% RSLogix 500 project PLCTEST_BAK000.RSS, saved by version 12.00.00.00 %
PROJECT "DRACO"    % processor: MicroLogix 1400 %

PROGRAM FILES
  LAD 2 "MAIN"  4 rungs
  LAD 3 "ALARM"  4 rungs
  LAD 4 "DIGITAL IO"  7 rungs
  LAD 5 "CONTROL"  6 rungs

DATA FILES
  O0 OUTPUT  7 elements
  I1 INPUT  10 elements
  S2 STATUS  66 elements
  B3 BINARY  1 elements
  T4 TIMER  3 elements
  C5 COUNTER  1 elements
  R6 CONTROL  1 elements
  N7 INTEGER  1 elements
  F8 FLOAT  1 elements

LADDER 2 "MAIN"
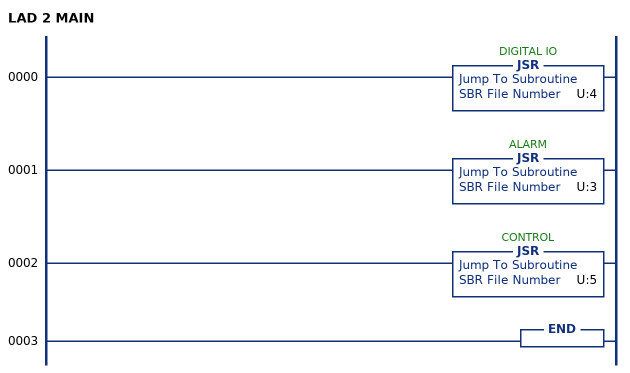
% Rung: 0 %
SOR JSR U:4 EOR
%   U:4  "DIGITAL IO" %
% Rung: 1 %
SOR JSR U:3 EOR
%   U:3  "ALARM" %
% Rung: 2 %
SOR JSR U:5 EOR
%   U:5  "CONTROL" %
% Rung: 3 %
SOR END EOR

LADDER 3 "ALARM"
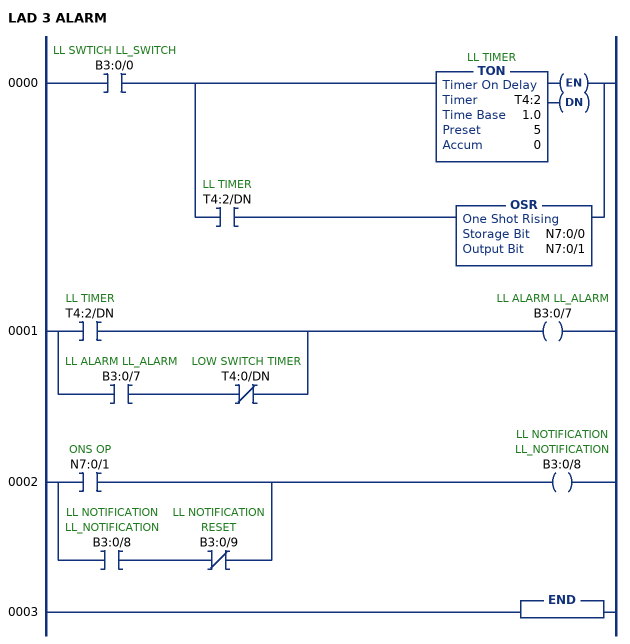
% Rung: 0 %
SOR XIC B3:0/0 BST TON T4:2 1.0 5 0 NXB XIC T4:2/DN OSR N7:0/0 N7:0/1 BND EOR
%   B3:0/0  LL_SWITCH  "LL SWTICH" %
%   T4:2  "LL TIMER" %
%   N7:0/1  "ONS OP" %
% Rung: 1 %
SOR BST XIC T4:2/DN NXB XIC B3:0/7 XIO T4:0/DN BND OTE B3:0/7 EOR
%   T4:2  "LL TIMER" %
%   B3:0/7  LL_ALARM  "LL ALARM" %
%   T4:0  "LOW SWITCH TIMER" %
% Rung: 2 %
SOR BST XIC N7:0/1 NXB XIC B3:0/8 XIO B3:0/9 BND OTE B3:0/8 EOR
%   N7:0/1  "ONS OP" %
%   B3:0/8  LL_NOTIFICATION  "LL NOTIFICATION" %
%   B3:0/9  "LL NOTIFICATION RESET" %
% Rung: 3 %
SOR END EOR

LADDER 4 "DIGITAL IO"
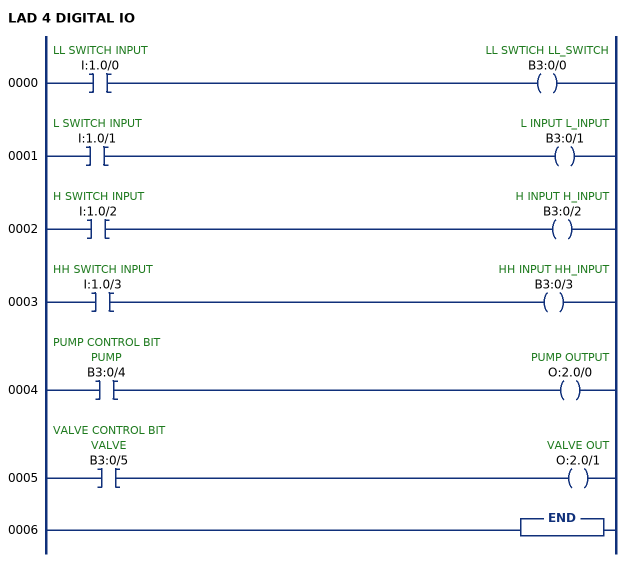
% Rung: 0 %
SOR XIC I:1.0/0 OTE B3:0/0 EOR
%   I:1.0/0  "LL SWITCH INPUT" %
%   B3:0/0  LL_SWITCH  "LL SWTICH" %
% Rung: 1 %
SOR XIC I:1.0/1 OTE B3:0/1 EOR
%   I:1.0/1  "L SWITCH INPUT" %
%   B3:0/1  L_INPUT  "L INPUT" %
% Rung: 2 %
SOR XIC I:1.0/2 OTE B3:0/2 EOR
%   I:1.0/2  "H SWITCH INPUT" %
%   B3:0/2  H_INPUT  "H INPUT" %
% Rung: 3 %
SOR XIC I:1.0/3 OTE B3:0/3 EOR
%   I:1.0/3  "HH SWITCH INPUT" %
%   B3:0/3  HH_INPUT  "HH INPUT" %
% Rung: 4 %
SOR XIC B3:0/4 OTE O:2.0/0 EOR
%   B3:0/4  PUMP  "PUMP CONTROL BIT" %
%   O:2.0/0  "PUMP OUTPUT" %
% Rung: 5 %
SOR XIC B3:0/5 OTE O:2.0/1 EOR
%   B3:0/5  VALVE  "VALVE CONTROL BIT" %
%   O:2.0/1  "VALVE OUT" %
% Rung: 6 %
SOR END EOR

LADDER 5 "CONTROL"
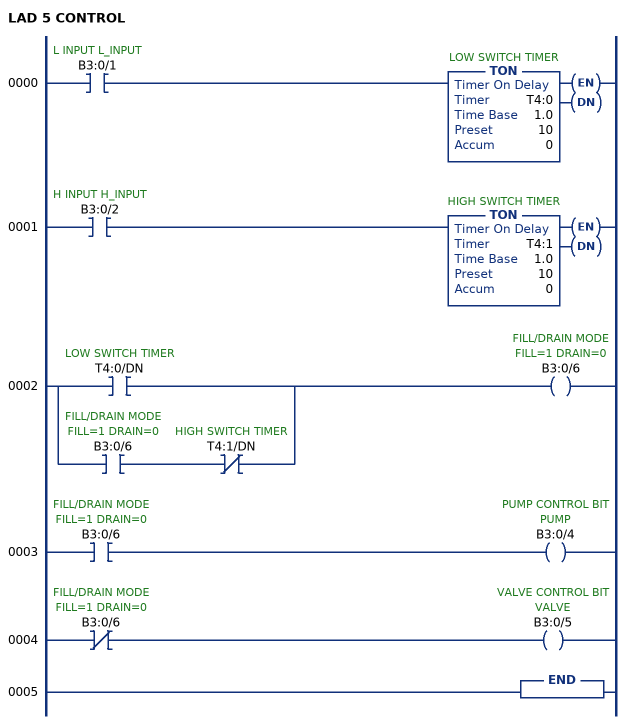
% Rung: 0 %
SOR XIC B3:0/1 TON T4:0 1.0 10 0 EOR
%   B3:0/1  L_INPUT  "L INPUT" %
%   T4:0  "LOW SWITCH TIMER" %
% Rung: 1 %
SOR XIC B3:0/2 TON T4:1 1.0 10 0 EOR
%   B3:0/2  H_INPUT  "H INPUT" %
%   T4:1  "HIGH SWITCH TIMER" %
% Rung: 2 %
SOR BST XIC T4:0/DN NXB XIC B3:0/6 XIO T4:1/DN BND OTE B3:0/6 EOR
%   T4:0  "LOW SWITCH TIMER" %
%   B3:0/6  "FILL/DRAIN MODE FILL=1 DRAIN=0" %
%   T4:1  "HIGH SWITCH TIMER" %
% Rung: 3 %
SOR XIC B3:0/6 OTE B3:0/4 EOR
%   B3:0/6  "FILL/DRAIN MODE FILL=1 DRAIN=0" %
%   B3:0/4  PUMP  "PUMP CONTROL BIT" %
% Rung: 4 %
SOR XIO B3:0/6 OTE B3:0/5 EOR
%   B3:0/6  "FILL/DRAIN MODE FILL=1 DRAIN=0" %
%   B3:0/5  VALVE  "VALVE CONTROL BIT" %
% Rung: 5 %
SOR END EOR

OTHER DOCUMENTED ADDRESSES
  N7:1  "ONS OB"

DATA TABLE (non-zero values as saved)
DATA T4
% .PRE .ACC %
% T4:0 % 10 0
% T4:1 % 10 0
% T4:2 % 5 0
